INTERFACE SocketA
VAR
	localAdr : T_AmsNetId;
	localPort : T_AmsPort;
END_VAR
VAR
	remoteAdr : T_AmsNetId;
	remotePort : T_AmsPort;
END_VAR

END_INTERFACE

(* stored: Version 1.1.0.1, ProductVersion 3.1.4024.11
   Itf SocketA: Id {2b29b4c7-983f-4531-8914-9a16bf207a39} *)
